// TIA Portal V19 export
DATA_BLOCK "MANUAL INTERLOCK DB"   // DB7
{ S7_Optimized_Access := 'TRUE' }
// stored: MemoryReserve 100
   VAR
      "MAIN ERROR" : Bool;
      "SYRUP MFG UNHEALTHY" : Int;
      "PREMIXING UNHEALTHY" : Int;
      "SUGAR UNHEALTHY" : Int;
      "MFG TRANSFER PROCESS INTERLOCK" : Int;
      "PREMIXING TRANSFER PROCESS INTERLOCK" : Int;
      "SUGAR TRANSFER PROCESS INTERLOCK" : Int;
   END_VAR
BEGIN
END_DATA_BLOCK
